{attribute 'GeneratedUsingTerminal: BK1250-0000-0019'}
{attribute addProperty BoxType "BK1250-0000-0019"}
{attribute addProperty Id "CouplerStateAT %I*UINT0"}
{attribute addProperty CRC "3424047604"}
{attribute addProperty Size "0"}
TYPE Inputs_CC16D1F4 EXTENDS TcoIo.InputBase_8311D824 :
STRUCT
	{attribute addProperty Name "CouplerState"}
	CouplerState AT %I* : UINT;
END_STRUCT
END_TYPE

(* stored: Version 1.2.0.0, ProductVersion 3.1.4024.9
   DUT Inputs_CC16D1F4: Id {66c4b537-8573-0c7c-0a94-b9c7d241cd42} *)
